Staubli VAL3: stop.pgx

program stop()
begin
  // Copyright (c) 2016, Ocado Technology - Robotics Research Team
  //
  // Licensed under the Apache License, Version 2.0 (the "License");
  // you may not use this file except in compliance with the License.
  // You may obtain a copy of the License at
  //
  //     http://www.apache.org/licenses/LICENSE-2.0
  //
  // Unless required by applicable law or agreed to in writing, software
  // distributed under the License is distributed on an "AS IS" BASIS,
  // WITHOUT WARRANTIES OR CONDITIONS OF ANY KIND, either express or implied.
  // See the License for the specific language governing permissions and
  // limitations under the License.

  // Reset robots motion
  resetMotion()
  // Show pop message with peding motion being cancelled
  popUpMsg("Pending movement commands have been cancelled.")

  // Clear user screen if library was loaded with success at the start program
  if nLibLoadError==0
    call libInterface:clearScreen()
  endIf

  // Kill running tasks
  taskKill(sTskMngTaskName)
  taskKill(sStreamTaskName)
  taskKill(sTrajPtTaskName)
  taskKill(sMotionTaskName)
  taskKill(sScreenTaskName)
  taskKill(sHtbtTaskName)
end
